FUNCTION_BLOCK "ModularAxis_Speed"   // FB5, LAD
{ S7_Optimized_Access := 'TRUE' }
// stored: MemoryReserve 100, SetENOAutomatically false
   VAR_INPUT
      HomingSensor : Bool;
      Reset : Bool;
      InverterOK : Bool;
      Axis : TO_SpeedAxis;
   END_VAR
   VAR_OUTPUT
      Status : "Status";
   END_VAR
   VAR_IN_OUT
      Execute : Bool;
      PositioningAxis : "S_SpeedAxis";
   END_VAR
   VAR
      State : "s_changeState";
      Delay { S7_SetPoint := 'True'} : "s_TON";
      PowerOff { S7_SetPoint := 'True'} : "s_TON";
      MC_POWER_Instance { ExternalAccessible := 'False'; ExternalVisible := 'False'; ExternalWritable := 'False'} : MC_POWER;
      MC_RESET_Instance { ExternalAccessible := 'False'; ExternalVisible := 'False'; ExternalWritable := 'False'} : MC_RESET;
      MC_HOME_Instance { ExternalAccessible := 'False'; ExternalVisible := 'False'; ExternalWritable := 'False'} : MC_HOME;
      MC_HALT_Instance { ExternalAccessible := 'False'; ExternalVisible := 'False'; ExternalWritable := 'False'} : MC_HALT;
      MC_MOVEJOG_Instance { ExternalAccessible := 'False'; ExternalVisible := 'False'; ExternalWritable := 'False'} : MC_MOVEJOG;
      R_TRIG_Homing { ExternalAccessible := 'False'; ExternalVisible := 'False'; ExternalWritable := 'False'} : R_TRIG;
      R_TRIG_HomeError { ExternalAccessible := 'False'; ExternalVisible := 'False'; ExternalWritable := 'False'} : R_TRIG;
      R_TRIG_HaltError { ExternalAccessible := 'False'; ExternalVisible := 'False'; ExternalWritable := 'False'} : R_TRIG;
      R_TRIG_PowerError { ExternalAccessible := 'False'; ExternalVisible := 'False'; ExternalWritable := 'False'} : R_TRIG;
      R_TRIG_JogError { ExternalAccessible := 'False'; ExternalVisible := 'False'; ExternalWritable := 'False'} : R_TRIG;
      R_TRIG_MoveRelError { ExternalAccessible := 'False'; ExternalVisible := 'False'; ExternalWritable := 'False'} : R_TRIG;
      R_TRIG_ResetError { ExternalAccessible := 'False'; ExternalVisible := 'False'; ExternalWritable := 'False'} : R_TRIG;
      F_TRIG_Inverter { ExternalAccessible := 'False'; ExternalVisible := 'False'; ExternalWritable := 'False'} : F_TRIG;
      Local : Struct
         HomingRequired : Bool;
         prevPosition : LReal;
      END_STRUCT;
   END_VAR
   VAR CONSTANT
      S_IDLE : Int := 10;
      S_HOME : Int := 20;
      S_STOP : Int := 30;
      S_ERROR : Int := 40;
      S_POWER_ON : Int := 50;
      S_MOVE_JOG : Int := 60;
      S_TEST : Int := 100;
      HOMING_ERROR : Word := 16#8000;
      HALT_ERROR : Word := 16#8001;
      POWER_ERROR : Word := 16#8002;
      JOG_ERROR : Word := 16#8003;
      MOVREL_ERROR : Word := 16#8004;
      RESET_ERROR : Word := 16#8005;
   END_VAR
BEGIN

REGION Network 1 (SCL)
   //************************************************************
   //===Author: Mateusz Połojko
   //-----Linkedin: https://pl.linkedin.com/in/mateusz-po%C5%82ojko-52a3541b1
   //-----Github: https://github.com/Bhazel95
   //===Description:
   //-----Motor control as to_speed axis
   //===Customer:
   //-----Apator Powogaz S.A.
   //************************************************************
END_REGION

REGION Network 2
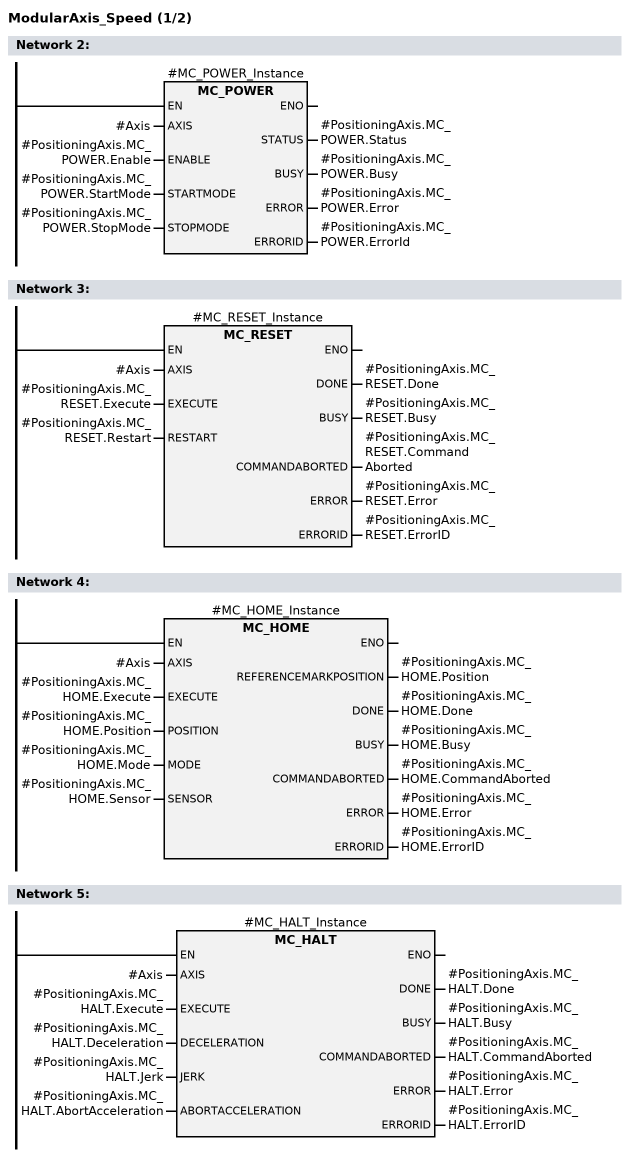
   RUNG wire#powerrail
      #MC_POWER_Instance.MC_POWER(Axis := #Axis, Enable := #PositioningAxis.MC_POWER.Enable, StartMode := #PositioningAxis.MC_POWER.StartMode, StopMode := #PositioningAxis.MC_POWER.StopMode, Status => #PositioningAxis.MC_POWER.Status, Busy => #PositioningAxis.MC_POWER.Busy, Error => #PositioningAxis.MC_POWER.Error, ErrorId => #PositioningAxis.MC_POWER.ErrorId)
   END_RUNG
   // the same network as SCL:
   #MC_POWER_Instance(Axis := #Axis,   // MC_POWER
                      Enable := #PositioningAxis.MC_POWER.Enable,
                      StartMode := #PositioningAxis.MC_POWER.StartMode,
                      StopMode := #PositioningAxis.MC_POWER.StopMode,
                      Status => #PositioningAxis.MC_POWER.Status,
                      Busy => #PositioningAxis.MC_POWER.Busy,
                      Error => #PositioningAxis.MC_POWER.Error,
                      ErrorId => #PositioningAxis.MC_POWER.ErrorId);
END_REGION

REGION Network 3
   RUNG wire#powerrail
      #MC_RESET_Instance.MC_RESET(Axis := #Axis, Execute := #PositioningAxis.MC_RESET.Execute, Restart := #PositioningAxis.MC_RESET.Restart, Done => #PositioningAxis.MC_RESET.Done, Busy => #PositioningAxis.MC_RESET.Busy, CommandAborted => #PositioningAxis.MC_RESET.CommandAborted, Error => #PositioningAxis.MC_RESET.Error, ErrorId => #PositioningAxis.MC_RESET.ErrorID)
   END_RUNG
   // the same network as SCL:
   #MC_RESET_Instance(Axis := #Axis,   // MC_RESET
                      Execute := #PositioningAxis.MC_RESET.Execute,
                      Restart := #PositioningAxis.MC_RESET.Restart,
                      Done => #PositioningAxis.MC_RESET.Done,
                      Busy => #PositioningAxis.MC_RESET.Busy,
                      CommandAborted => #PositioningAxis.MC_RESET.CommandAborted,
                      Error => #PositioningAxis.MC_RESET.Error,
                      ErrorId => #PositioningAxis.MC_RESET.ErrorID);
END_REGION

REGION Network 4
   RUNG wire#powerrail
      #MC_HOME_Instance.MC_HOME(Axis := #Axis, Execute := #PositioningAxis.MC_HOME.Execute, Position := #PositioningAxis.MC_HOME.Position, Mode := #PositioningAxis.MC_HOME.Mode, Sensor := #PositioningAxis.MC_HOME.Sensor, ReferenceMarkPosition => #PositioningAxis.MC_HOME.Position, Done => #PositioningAxis.MC_HOME.Done, Busy => #PositioningAxis.MC_HOME.Busy, CommandAborted => #PositioningAxis.MC_HOME.CommandAborted, Error => #PositioningAxis.MC_HOME.Error, ErrorId => #PositioningAxis.MC_HOME.ErrorID)
   END_RUNG
   // the same network as SCL:
   #MC_HOME_Instance(Axis := #Axis,   // MC_HOME
                     Execute := #PositioningAxis.MC_HOME.Execute,
                     Position := #PositioningAxis.MC_HOME.Position,
                     Mode := #PositioningAxis.MC_HOME.Mode,
                     Sensor := #PositioningAxis.MC_HOME.Sensor,
                     ReferenceMarkPosition => #PositioningAxis.MC_HOME.Position,
                     Done => #PositioningAxis.MC_HOME.Done,
                     Busy => #PositioningAxis.MC_HOME.Busy,
                     CommandAborted => #PositioningAxis.MC_HOME.CommandAborted,
                     Error => #PositioningAxis.MC_HOME.Error,
                     ErrorId => #PositioningAxis.MC_HOME.ErrorID);
END_REGION

REGION Network 5
   RUNG wire#powerrail
      #MC_HALT_Instance.MC_HALT(Axis := #Axis, Execute := #PositioningAxis.MC_HALT.Execute, Deceleration := #PositioningAxis.MC_HALT.Deceleration, Jerk := #PositioningAxis.MC_HALT.Jerk, AbortAcceleration := #PositioningAxis.MC_HALT.AbortAcceleration, Done => #PositioningAxis.MC_HALT.Done, Busy => #PositioningAxis.MC_HALT.Busy, CommandAborted => #PositioningAxis.MC_HALT.CommandAborted, Error => #PositioningAxis.MC_HALT.Error, ErrorId => #PositioningAxis.MC_HALT.ErrorID)
   END_RUNG
   // the same network as SCL:
   #MC_HALT_Instance(Axis := #Axis,   // MC_HALT
                     Execute := #PositioningAxis.MC_HALT.Execute,
                     Deceleration := #PositioningAxis.MC_HALT.Deceleration,
                     Jerk := #PositioningAxis.MC_HALT.Jerk,
                     AbortAcceleration := #PositioningAxis.MC_HALT.AbortAcceleration,
                     Done => #PositioningAxis.MC_HALT.Done,
                     Busy => #PositioningAxis.MC_HALT.Busy,
                     CommandAborted => #PositioningAxis.MC_HALT.CommandAborted,
                     Error => #PositioningAxis.MC_HALT.Error,
                     ErrorId => #PositioningAxis.MC_HALT.ErrorID);
END_REGION

REGION Network 6
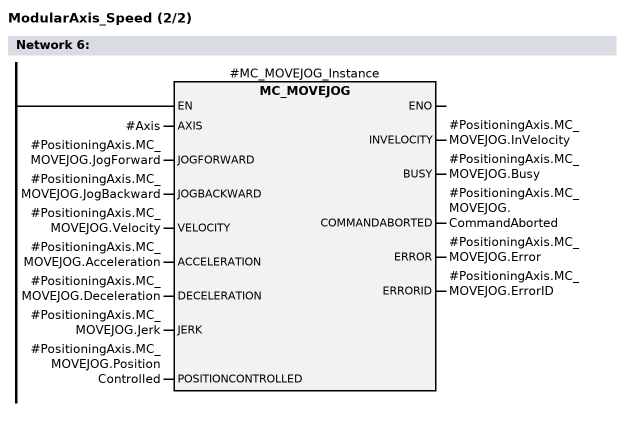
   RUNG wire#powerrail
      #MC_MOVEJOG_Instance.MC_MOVEJOG(Axis := #Axis, JogForward := #PositioningAxis.MC_MOVEJOG.JogForward, JogBackward := #PositioningAxis.MC_MOVEJOG.JogBackward, Velocity := #PositioningAxis.MC_MOVEJOG.Velocity, Acceleration := #PositioningAxis.MC_MOVEJOG.Acceleration, Deceleration := #PositioningAxis.MC_MOVEJOG.Deceleration, Jerk := #PositioningAxis.MC_MOVEJOG.Jerk, PositionControlled := #PositioningAxis.MC_MOVEJOG.PositionControlled, InVelocity => #PositioningAxis.MC_MOVEJOG.InVelocity, Busy => #PositioningAxis.MC_MOVEJOG.Busy, CommandAborted => #PositioningAxis.MC_MOVEJOG.CommandAborted, Error => #PositioningAxis.MC_MOVEJOG.Error, ErrorId => #PositioningAxis.MC_MOVEJOG.ErrorID)
   END_RUNG
   // the same network as SCL:
   #MC_MOVEJOG_Instance(Axis := #Axis,   // MC_MOVEJOG
                        JogForward := #PositioningAxis.MC_MOVEJOG.JogForward,
                        JogBackward := #PositioningAxis.MC_MOVEJOG.JogBackward,
                        Velocity := #PositioningAxis.MC_MOVEJOG.Velocity,
                        Acceleration := #PositioningAxis.MC_MOVEJOG.Acceleration,
                        Deceleration := #PositioningAxis.MC_MOVEJOG.Deceleration,
                        Jerk := #PositioningAxis.MC_MOVEJOG.Jerk,
                        PositionControlled := #PositioningAxis.MC_MOVEJOG.PositionControlled,
                        InVelocity => #PositioningAxis.MC_MOVEJOG.InVelocity,
                        Busy => #PositioningAxis.MC_MOVEJOG.Busy,
                        CommandAborted => #PositioningAxis.MC_MOVEJOG.CommandAborted,
                        Error => #PositioningAxis.MC_MOVEJOG.Error,
                        ErrorId => #PositioningAxis.MC_MOVEJOG.ErrorID);
END_REGION

REGION Network 8 (SCL)
   REGION R/F Trigs
       #F_TRIG_Inverter(CLK := #InverterOK);
       #R_TRIG_HomeError(CLK := #PositioningAxis.MC_HOME.Error);
       #R_TRIG_HaltError(CLK := #PositioningAxis.MC_HALT.Error);
       #R_TRIG_PowerError(CLK := #PositioningAxis.MC_POWER.Error);
       #R_TRIG_JogError(CLK := #PositioningAxis.MC_MOVEJOG.Error);
      // #R_TRIG_MoveRelError(CLK := #PositioningAxis.MC_MOVERELATIVE.Error);
       #R_TRIG_ResetError(CLK := #PositioningAxis.MC_RESET.Error);
       #R_TRIG_Homing(CLK := #HomingSensor);

   END_REGION
   #Delay.PT := T#500MS;
   #Delay.Timer(IN := #Delay.IN,
                PT := #Delay.PT);
   #PowerOff.PT := T#180S;
   #PowerOff.Timer(IN := #PowerOff.IN,
                   PT := #PowerOff.PT);

   CASE #State.state OF
       #S_IDLE:
           //Funkcja wejścia
           IF #State.inputFlag AND NOT #State.outputFlag THEN
               #Execute := FALSE;
               #State.name := 'IDLE';
               #Status.Busy := FALSE;
               #Status.Ready := TRUE;
               // #Status.Done := FALSE;
               #Status.Error := FALSE;
               #PowerOff.IN := TRUE;
           END_IF;

           //Funkcja cykliczna
           IF NOT #State.inputFlag AND NOT #State.outputFlag THEN
               IF #PowerOff.Timer.Q THEN
                   #PositioningAxis.MC_POWER.Enable := FALSE;
               END_IF;
               IF #Reset THEN
                   // Statement section IF
                   ;
               END_IF;


               IF #Execute THEN
                   IF #PositioningAxis.MC_POWER.Status THEN
                       "changeState"(newState := #S_MOVE_JOG,
                                     Data := #State);
                   ELSE
                       #PositioningAxis.MC_POWER.Enable := FALSE;
                       "changeState"(newState := #S_POWER_ON,
                                     Data := #State);
                   END_IF;
               END_IF;
               IF #PositioningAxis.MC_MOVEJOG.JogForward OR #PositioningAxis.MC_MOVEJOG.JogBackward THEN
                   #Status.Done := FALSE;
                   #Status.Busy := TRUE;
                   //#Local.HomingRequired := TRUE;
               END_IF;
           END_IF;

           //Funkcja wyjściowa 
           IF #State.outputFlag THEN
               #PowerOff.IN := FALSE;
               #Status.Busy := TRUE;
           END_IF;

       #S_HOME:
           //Funkcja wejścia
           IF #State.inputFlag AND NOT #State.outputFlag THEN
               #State.name := 'HOMING';
               #Status.Busy := TRUE;
               #Status.Ready := FALSE;
               #Status.Done := FALSE;
               #Status.Error := FALSE;
               #PositioningAxis.MC_HOME.Mode := 8;
               #PositioningAxis.MC_HOME.Execute := TRUE;
           END_IF;

           //Funkcja cykliczna
           IF NOT #State.inputFlag AND NOT #State.outputFlag THEN
               IF #PositioningAxis.MC_HOME.Done THEN
                   #Local.HomingRequired := FALSE;
                   #Status.Done := TRUE;
                   "changeState"(newState := #S_IDLE,
                                 Data := #State);
               END_IF;
           END_IF;

           //Funkcja wyjściowa 
           IF #State.outputFlag THEN
               #PositioningAxis.MC_HOME.Execute := FALSE;
           END_IF;

       #S_ERROR:
           //Funkcja wejścia
           IF #State.inputFlag AND NOT #State.outputFlag THEN
               #State.name := 'ERROR';
               #Status.Busy := FALSE;
               #Status.Ready := FALSE;
               #Status.Done := FALSE;
               #Status.Error := TRUE;
               //#Local.HomingRequired := TRUE;
               #PositioningAxis.MC_HOME.Execute := FALSE;
               #PositioningAxis.MC_POWER.Enable := FALSE;
              // #PositioningAxis.MC_MOVERELATIVE.Execute := FALSE;
               #PositioningAxis.MC_HALT.Execute := FALSE;
               #PositioningAxis.MC_RESET.Execute := FALSE;
               #PositioningAxis.MC_MOVEJOG.JogBackward := FALSE;
               #PositioningAxis.MC_MOVEJOG.JogForward := FALSE;
           END_IF;

           //Funkcja cykliczna
           IF NOT #State.inputFlag AND NOT #State.outputFlag THEN
               IF #Reset THEN
                   // #MC_RESET_Instance.Restart := FALSE;
                   #PositioningAxis.MC_RESET.Execute := TRUE;
               END_IF;
               IF #PositioningAxis.MC_RESET.Done AND #InverterOK THEN
                   "changeState"(newState := #S_POWER_ON,
                                 Data := #State);
               END_IF;
           END_IF;

           //Funkcja wyjściowa 
           IF #State.outputFlag THEN
               #Status.Error := FALSE;
               #Status.Busy := TRUE;
               #PositioningAxis.MC_RESET.Execute := FALSE;
           END_IF;

       #S_POWER_ON:
           //Funkcja wejścia
           IF #State.inputFlag AND NOT #State.outputFlag THEN
               #State.name := 'ERROR';
               #Status.Busy := TRUE;
               #Status.Ready := FALSE;
               #Status.Done := FALSE;
               #Status.Error := FALSE;
               #PositioningAxis.MC_POWER.Enable := TRUE;
           END_IF;

           //Funkcja cykliczna
           IF NOT #State.inputFlag AND NOT #State.outputFlag THEN
               IF #PositioningAxis.MC_POWER.Status THEN
                   "changeState"(newState := #S_IDLE,
                                 Data := #State);
               END_IF;
           END_IF;

           //Funkcja wyjściowa 
           IF #State.outputFlag THEN
               ;
           END_IF;

       #S_MOVE_JOG:
           //Funkcja wejścia
           IF #State.inputFlag AND NOT #State.outputFlag THEN
               #State.name := 'MOVING';
               #Status.Busy := TRUE;
               #Status.Ready := FALSE;
               #Status.Done := FALSE;
               #Status.Error := FALSE;
               //#Local.prevPosition := #Axis.ActualPosition;
               #PositioningAxis.MC_MOVEJOG.Acceleration := 0.3;
               #PositioningAxis.MC_MOVEJOG.Deceleration := 0.7;
               #PositioningAxis.MC_MOVEJOG.Velocity := 0.15;
               #PositioningAxis.MC_MOVEJOG.JogBackward := FALSE;
               #PositioningAxis.MC_MOVEJOG.JogForward := TRUE;
               #Delay.IN := FALSE;
           END_IF;

           //Funkcja cykliczna
           IF NOT #State.inputFlag AND NOT #State.outputFlag THEN
               IF #R_TRIG_Homing.Q THEN
                   #Status.Done := TRUE;
                   #PositioningAxis.MC_MOVEJOG.JogBackward := FALSE;
                   #PositioningAxis.MC_MOVEJOG.JogForward := FALSE;
                   #Delay.IN := TRUE;
               END_IF;
               IF #Delay.Timer.Q THEN

                   "changeState"(newState := #S_IDLE,
                                 Data := #State);
               END_IF;

           END_IF;

           //Funkcja wyjściowa 
           IF #State.outputFlag THEN
               #Delay.IN := FALSE;
           END_IF;

       #S_TEST:
           ;
   END_CASE;

   IF #R_TRIG_HomeError.Q THEN
       #Status.ErrorStatus := #HOMING_ERROR;
       "changeState"(newState := #S_ERROR,
                     Data := #State);
   ELSIF #R_TRIG_HaltError.Q THEN
       #Status.ErrorStatus := #HALT_ERROR;
       "changeState"(newState := #S_ERROR,
                     Data := #State);
   ELSIF #R_TRIG_JogError.Q THEN
       #Status.ErrorStatus := #JOG_ERROR;
       "changeState"(newState := #S_ERROR,
                     Data := #State);
   ELSIF #R_TRIG_MoveRelError.Q THEN
       #Status.ErrorStatus := #MOVREL_ERROR;
       "changeState"(newState := #S_ERROR,
                     Data := #State);
   ELSIF #R_TRIG_PowerError.Q THEN
       #Status.ErrorStatus := #POWER_ERROR;
       "changeState"(newState := #S_ERROR,
                     Data := #State);
   ELSIF #R_TRIG_ResetError.Q THEN
       #Status.ErrorStatus := #RESET_ERROR;
       "changeState"(newState := #S_ERROR,
                     Data := #State);
   END_IF;

   IF #F_TRIG_Inverter.Q THEN
       "changeState"(newState := #S_ERROR,
                     Data := #State);
   END_IF;

   IF NOT "DEV_7".Convoyer.Modular_A.Sensors.JogBack THEN
       #PositioningAxis.MC_MOVEJOG.JogBackward := FALSE;
   END_IF;

   REGION Change state
       IF #State.inputFlag AND NOT #State.outputFlag THEN
           #State.inputFlag := FALSE;
       END_IF;
       #State.outputFlag := FALSE;
   END_REGION
END_REGION
END_FUNCTION_BLOCK

FUNCTION "FC_008_OPC" : Void
{ S7_Optimized_Access := 'TRUE' }
VERSION : 0.1

BEGIN
END_FUNCTION

FUNCTION "FC_09_HMI" : Void
{ S7_Optimized_Access := 'TRUE' }
VERSION : 0.1

BEGIN
	//************************************************************
	//===Author: Mateusz Połojko
	//-----Linkedin: https://pl.linkedin.com/in/mateusz-po%C5%82ojko-52a3541b1
	//-----Github: https://github.com/Bhazel95
	//===Description:
	//-----HMI assigments
	//===Customer:
	//-----Apator Powogaz S.A.
	//************************************************************
	
	REGION Camera state  
	    "DEV_7".Convoyer.Modular_A.HMI.Camera.State := "ModularConvoyer_7A_DB".CameraConnectionTCP_Instance.State.name;
	    "DEV_7".Convoyer.Modular_B.HMI.Camera.State := "ModularConvoyer_7B_DB".CameraConnectionTCP_Instance.State.name;
	    "DEV_10".Convoyer.Modular_A.HMI.Camera.State := "ModularConvoyer_10A_DB".CameraConnectionTCP_Instance.State.name;
	END_REGION
	
END_FUNCTION

FUNCTION "FC_010_Outputs" : Void
{ S7_Optimized_Access := 'TRUE' }
VERSION : 0.1

BEGIN
	//************************************************************
	//===Author: Mateusz Połojko
	//-----Linkedin: https://pl.linkedin.com/in/mateusz-po%C5%82ojko-52a3541b1
	//-----Github: https://github.com/Bhazel95
	//===Description:
	//-----Hardware output assigment
	//===Customer:
	//-----Apator Powogaz S.A.
	//************************************************************
	
	REGION 7A
	    REGION Button box left
	        "7A_BUTTON_LIGHT_START_1" := "DEV_7".Convoyer.Modular_A.ButtonControl.ButtonBoxLeft.LightStart;
	        "7A_BUTTON_LIGHT_RESET_1" := "DEV_7".Convoyer.Modular_A.ButtonControl.ButtonBoxLeft.LightReset;
	        "7A_BUTTON_LIGHT_STOP_1" := "DEV_7".Convoyer.Modular_A.ButtonControl.ButtonBoxLeft.LightStop;
	        "7A_BUTTON_LIGHT_ESTOP_1" := NOT "7A_ESTOP_1";
	    END_REGION
	    REGION Button box right
	        "7A_BUTTON_LIGHT_START_2" := "DEV_7".Convoyer.Modular_A.ButtonControl.ButtonBoxRight.LightStart;
	        "7A_BUTTON_LIGHT_RESET_2" := "DEV_7".Convoyer.Modular_A.ButtonControl.ButtonBoxRight.LightReset;
	        "7A_BUTTON_LIGHT_STOP_2" := "DEV_7".Convoyer.Modular_A.ButtonControl.ButtonBoxRight.LightStop;
	        "7A_BUTTON_LIGHT_ESTOP_2" := NOT "7A_ESTOP_2";
	    END_REGION
	    REGION Lights    
	        "7A_LIGHTS_BUZZER_1" := "DEV_7".Convoyer.Modular_A.Lights.Blue;
	        "7A_LIGHTS_GREEN_1" := "DEV_7".Convoyer.Modular_A.Lights.Green;
	        "7A_LIGHTS_RED_1" := "DEV_7".Convoyer.Modular_A.Lights.Red;
	        "7A_LIGHTS_ORANGE_1" := "DEV_7".Convoyer.Modular_A.Lights.Orange;
	    END_REGION
	    REGION Pneumatics
	        "7A_VALVE_IN_1" := "DEV_7".Convoyer.Modular_A.Pneumatics.Stamping.Coils.In;
	        "7A_VALVE_OUT_1" := "DEV_7".Convoyer.Modular_A.Pneumatics.Stamping.Coils.Out;
	        
	        "7A_VALVE_IN_2" := "DEV_7".Convoyer.Modular_A.Pneumatics.Valve.Coils.In;
	        "7A_VALVE_OUT_2" := "DEV_7".Convoyer.Modular_A.Pneumatics.Valve.Coils.Out;
	        
	        IF "DEV_7".Convoyer.Modular_A.Safety.SafetyOK AND "DEV_7".Convoyer.Modular_A.Sensors.Span THEN
	            "DEV_7".Convoyer.Modular_A.Pneumatics.IVT.Sensor.Scaled.SetNorm := NORM_X(MIN := 0, VALUE := "DEV_7".Convoyer.Modular_A.Pneumatics.IVT.Sensor.Analog.SetValue, MAX := 7);
	            "7A_IVT_OutputSignal_1" := SCALE_X(MIN := 0, VALUE := "DEV_7".Convoyer.Modular_A.Pneumatics.IVT.Sensor.Scaled.SetNorm, MAX := 32767);
	        ELSE
	            "DEV_7".Convoyer.Modular_A.Pneumatics.IVT.Sensor.Scaled.SetNorm := NORM_X(MIN := 0.0, VALUE := 0.0, MAX := 7);
	            "7A_IVT_OutputSignal_1" := SCALE_X(MIN := 0, VALUE := "DEV_7".Convoyer.Modular_A.Pneumatics.IVT.Sensor.Scaled.SetNorm, MAX := 32767);
	        END_IF;
	    END_REGION
	END_REGION
	REGION 7B
	    REGION Button box left
	        "7B_BUTTON_LIGHT_START_1" := "DEV_7".Convoyer.Modular_B.ButtonControl.ButtonBoxLeft.LightStart;
	        "7B_BUTTON_LIGHT_RESET_1" := "DEV_7".Convoyer.Modular_B.ButtonControl.ButtonBoxLeft.LightReset;
	        "7B_BUTTON_LIGHT_STOP_1" := "DEV_7".Convoyer.Modular_B.ButtonControl.ButtonBoxLeft.LightStop;
	        "7B_BUTTON_LIGHT_ESTOP_1" := NOT "7B_ESTOP_1";
	    END_REGION
	    REGION Button box right
	        "7B_BUTTON_LIGHT_START_2" := "DEV_7".Convoyer.Modular_B.ButtonControl.ButtonBoxRight.LightStart;
	        "7B_BUTTON_LIGHT_RESET_2" := "DEV_7".Convoyer.Modular_B.ButtonControl.ButtonBoxRight.LightReset;
	        "7B_BUTTON_LIGHT_STOP_2" := "DEV_7".Convoyer.Modular_B.ButtonControl.ButtonBoxRight.LightStop;
	        "7B_BUTTON_LIGHT_ESTOP_2" := NOT "7B_ESTOP_2";
	    END_REGION
	    REGION Lights    
	        "7B_LIGHTS_BUZZER_1" := "DEV_7".Convoyer.Modular_B.Lights.Blue;
	        "7B_LIGHTS_GREEN_1" := "DEV_7".Convoyer.Modular_B.Lights.Green;
	        "7B_LIGHTS_RED_1" := "DEV_7".Convoyer.Modular_B.Lights.Red;
	        "7B_LIGHTS_ORANGE_1" := "DEV_7".Convoyer.Modular_B.Lights.Orange;
	    END_REGION
	    REGION Pneumatics
	        "7B_VALVE_IN_2" := "DEV_7".Convoyer.Modular_B.Pneumatics.Stamping.Coils.In;
	        "7B_VALVE_OUT_2" := "DEV_7".Convoyer.Modular_B.Pneumatics.Stamping.Coils.Out;
	        
	        "7B_VALVE_IN_1" := "DEV_7".Convoyer.Modular_B.Pneumatics.Valve.Coils.In;
	        "7B_VALVE_OUT_1" := "DEV_7".Convoyer.Modular_B.Pneumatics.Valve.Coils.Out;
	        
	        IF "DEV_7".Convoyer.Modular_B.Safety.SafetyOK AND "DEV_7".Convoyer.Modular_B.Sensors.Span THEN
	            "DEV_7".Convoyer.Modular_B.Pneumatics.IVT.Sensor.Scaled.SetNorm := NORM_X(MIN := 0, VALUE := "DEV_7".Convoyer.Modular_B.Pneumatics.IVT.Sensor.Analog.SetValue, MAX := 7);
	            "7B_IVT_OutputSignal_1" := SCALE_X(MIN := 0, VALUE := "DEV_7".Convoyer.Modular_B.Pneumatics.IVT.Sensor.Scaled.SetNorm, MAX := 32767);
	        ELSE
	            "DEV_7".Convoyer.Modular_B.Pneumatics.IVT.Sensor.Scaled.SetNorm := NORM_X(MIN := 0.0, VALUE := 0.0, MAX := 7);
	            "7B_IVT_OutputSignal_1" := SCALE_X(MIN := 0, VALUE := "DEV_7".Convoyer.Modular_B.Pneumatics.IVT.Sensor.Scaled.SetNorm, MAX := 32767);
	        END_IF;
	    END_REGION
	END_REGION
	REGION Main Cabinet
	    "7_BUTTON_LIGHT_RESET_6" := "DEV_7".Convoyer.Modular_A.ButtonControl.CabinetBox.LightReset OR "DEV_7".Convoyer.Modular_B.ButtonControl.CabinetBox.LightReset;
	    "7_BUTTON_LIGHT_ESTOP_6" := NOT "7_ESTOP";
	END_REGION
	REGION 24V Main Cabinet
	    "7AB_24V_OK" := "7_24V_OK";
	END_REGION
	
	
	REGION 10A
	    REGION Button box left
	        "10A_BUTTON_LIGHT_START_1" := "DEV_10".Convoyer.Modular_A.ButtonControl.ButtonBoxLeft.LightStart;
	        "10A_BUTTON_LIGHT_RESET_1" := "DEV_10".Convoyer.Modular_A.ButtonControl.ButtonBoxLeft.LightReset;
	        "10A_BUTTON_LIGHT_STOP_1" := "DEV_10".Convoyer.Modular_A.ButtonControl.ButtonBoxLeft.LightStop;
	        "10A_BUTTON_LIGHT_ESTOP_1" := NOT "10A_ESTOP_1";
	    END_REGION
	    REGION Button box right
	        "10A_BUTTON_LIGHT_START_2" := "DEV_10".Convoyer.Modular_A.ButtonControl.ButtonBoxRight.LightStart;
	        "10A_BUTTON_LIGHT_RESET_2" := "DEV_10".Convoyer.Modular_A.ButtonControl.ButtonBoxRight.LightReset;
	        "10A_BUTTON_LIGHT_STOP_2" := "DEV_10".Convoyer.Modular_A.ButtonControl.ButtonBoxRight.LightStop;
	        "10A_BUTTON_LIGHT_ESTOP_2" := NOT "10A_ESTOP_2";
	    END_REGION
	    REGION Lights    
	        "10A_LIGHTS_BUZZER_1" := "DEV_10".Convoyer.Modular_A.Lights.Blue;
	        "10A_LIGHTS_GREEN_1" := "DEV_10".Convoyer.Modular_A.Lights.Green;
	        "10A_LIGHTS_RED_1" := "DEV_10".Convoyer.Modular_A.Lights.Red;
	        "10A_LIGHTS_ORANGE_1" := "DEV_10".Convoyer.Modular_A.Lights.Orange;
	    END_REGION
	    REGION Pneumatics
	        "10A_VALVE_IN_1" := "DEV_10".Convoyer.Modular_A.Pneumatics.Stamping.Coils.In;
	        "10A_VALVE_OUT_1" := "DEV_10".Convoyer.Modular_A.Pneumatics.Stamping.Coils.Out;
	        
	        "10A_VALVE_IN_2" := "DEV_10".Convoyer.Modular_A.Pneumatics.Valve.Coils.In;
	        "10A_VALVE_OUT_2" := "DEV_10".Convoyer.Modular_A.Pneumatics.Valve.Coils.Out;
	        
	        IF "DEV_10".Convoyer.Modular_A.Safety.SafetyOK AND "DEV_10".Convoyer.Modular_A.Sensors.Span THEN
	            "DEV_10".Convoyer.Modular_A.Pneumatics.IVT.Sensor.Scaled.SetNorm := NORM_X(MIN := 0, VALUE := "DEV_10".Convoyer.Modular_A.Pneumatics.IVT.Sensor.Analog.SetValue, MAX := 7);
	            "10A_IVT_OutputSignal_1" := SCALE_X(MIN := 0, VALUE := "DEV_10".Convoyer.Modular_A.Pneumatics.IVT.Sensor.Scaled.SetNorm, MAX := 32767);
	        ELSE
	            "DEV_10".Convoyer.Modular_A.Pneumatics.IVT.Sensor.Scaled.SetNorm := NORM_X(MIN := 0.0, VALUE := 0.0, MAX := 7);
	            "10A_IVT_OutputSignal_1" := SCALE_X(MIN := 0, VALUE := "DEV_10".Convoyer.Modular_A.Pneumatics.IVT.Sensor.Scaled.SetNorm, MAX := 32767);
	        END_IF;
	    END_REGION
	END_REGION
	REGION 10 Cabinet
	    //dla 10b dodac or 10b
	    "10_BUTTON_LIGHT_RESET_6" := "DEV_10".Convoyer.Modular_A.ButtonControl.CabinetBox.LightReset;
	    "10_BUTTON_LIGHT_ESTOP_6" := NOT "10_ESTOP";
	END_REGION
	//Do zmiany
	REGION 24V 10 Cabinet  
	    "10AB_24V_OK" := TRUE;
	END_REGION
	
END_FUNCTION

FUNCTION_BLOCK "CabinetDiagReset_10"   // FB13, F_LAD
{ S7_Optimized_Access := 'TRUE' }
   VAR_INPUT
      RESET : Bool;
   END_VAR
BEGIN

REGION Network 1: 1=Acknowledgment for reintegration
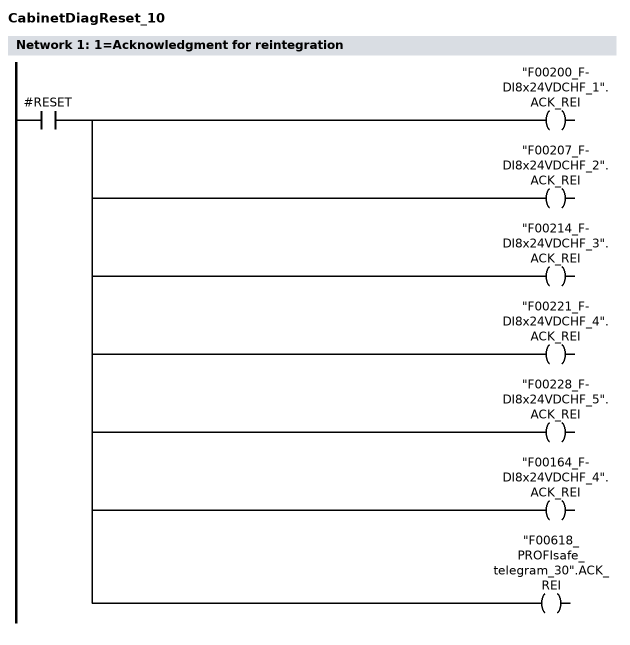
   RUNG wire#powerrail
      Contact( #RESET )
      wire#w1
      Coil( "F00200_F-DI8x24VDCHF_1".ACK_REI )
   END_RUNG
   RUNG wire#w1
      Coil( "F00207_F-DI8x24VDCHF_2".ACK_REI )
   END_RUNG
   RUNG wire#w1
      Coil( "F00214_F-DI8x24VDCHF_3".ACK_REI )
   END_RUNG
   RUNG wire#w1
      Coil( "F00221_F-DI8x24VDCHF_4".ACK_REI )
   END_RUNG
   RUNG wire#w1
      Coil( "F00228_F-DI8x24VDCHF_5".ACK_REI )
   END_RUNG
   RUNG wire#w1
      Coil( "F00164_F-DI8x24VDCHF_4".ACK_REI )
   END_RUNG
   RUNG wire#w1
      Coil( "F00618_PROFIsafe_telegram_30".ACK_REI )
   END_RUNG
   // the same network as SCL:
   "F00200_F-DI8x24VDCHF_1".ACK_REI := #RESET;
   "F00207_F-DI8x24VDCHF_2".ACK_REI := #RESET;
   "F00214_F-DI8x24VDCHF_3".ACK_REI := #RESET;
   "F00221_F-DI8x24VDCHF_4".ACK_REI := #RESET;
   "F00228_F-DI8x24VDCHF_5".ACK_REI := #RESET;
   "F00164_F-DI8x24VDCHF_4".ACK_REI := #RESET;
   "F00618_PROFIsafe_telegram_30".ACK_REI := #RESET;
END_REGION
END_FUNCTION_BLOCK

FUNCTION_BLOCK "Convoyer7"   // FB6, F_LAD
{ S7_Optimized_Access := 'TRUE' }
   VAR_INPUT
      InverterStatus : "LDrvSafe_typeSinaTlg30Status";
      ESTOP : Bool;
      LIGHT_CURTAIN : Bool;
      PROCES_STAMPING : Bool;
      DOOR : Bool;
      FRQ_FEEDBACK : Bool;
      RESET : Bool;
   END_VAR
   VAR_OUTPUT
      InverterControl : "LDrvSafe_typeSinaTlg30Control";
      SAFETY_OK : Bool;
      INVERTER_OK : Bool;
      FRQ_NOK : Bool;
      REQ_RESET_ESTOP : Bool;
      SAFETY_VALVE : Bool;
   END_VAR
   VAR
      ESTOP_ON : Bool;
      INVERTER_FAULT : Bool;
      ESTOP1_Instance : ESTOP1;
      LDrvSafe_SinaTlg30Control_Instance : "LDrvSafe_SinaTlg30Control";
      LDrvSafe_SinaTlg30Status_Instance : "LDrvSafe_SinaTlg30Status";
   END_VAR
BEGIN

REGION Network 1
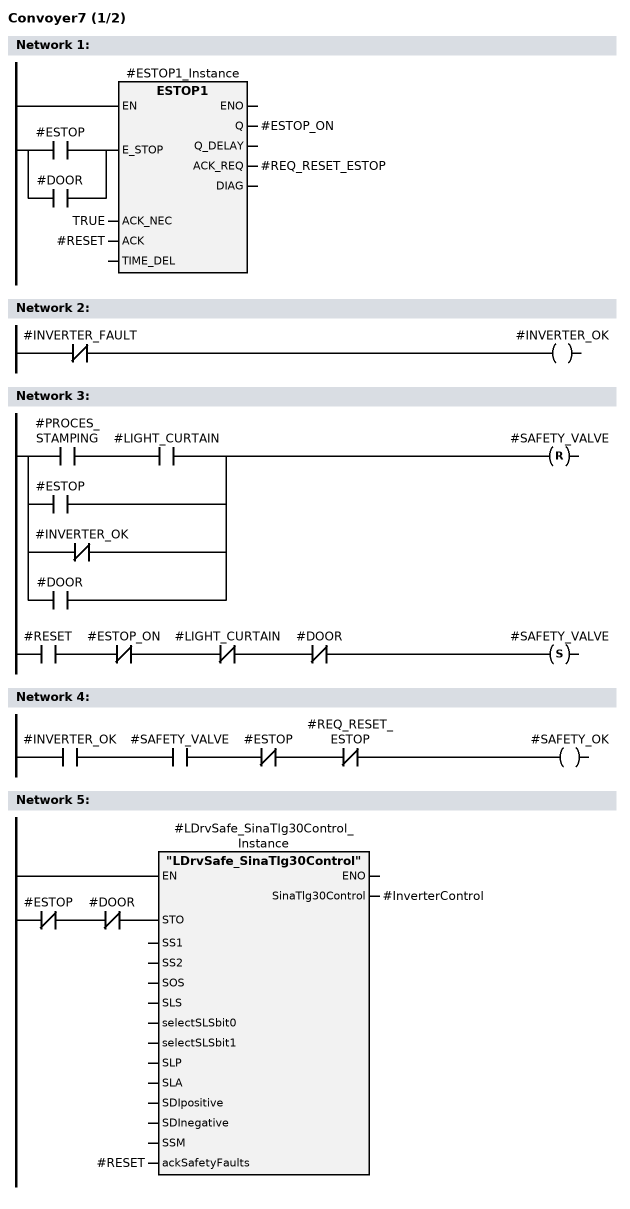
   RUNG wire#powerrail
      #ESTOP1_Instance.ESTOP1(E_STOP := wire#w1, ACK_NEC := TRUE, ACK := #RESET, TIME_DEL :=, Q => #ESTOP_ON, Q_DELAY =>, ACK_REQ => #REQ_RESET_ESTOP, DIAG =>)
   END_RUNG
   RUNG wire#powerrail
      Contact( #ESTOP )
   END_RUNG wire#w1
   RUNG wire#powerrail
      Contact( #DOOR )
   END_RUNG wire#w1
   // the same network as SCL:
   #ESTOP1_Instance(E_STOP := #ESTOP OR #DOOR,   // ESTOP1
                    ACK_NEC := TRUE,
                    ACK := #RESET,
                    Q => #ESTOP_ON,
                    ACK_REQ => #REQ_RESET_ESTOP);
END_REGION

REGION Network 2
   RUNG wire#powerrail
      I_Contact( #INVERTER_FAULT )
      Coil( #INVERTER_OK )
   END_RUNG
   // the same network as SCL:
   #INVERTER_OK := NOT #INVERTER_FAULT;
END_REGION

REGION Network 3
   RUNG wire#powerrail
      Contact( #PROCES_STAMPING )
      Contact( #LIGHT_CURTAIN )
      wire#w1
      R_Coil( #SAFETY_VALVE )
   END_RUNG
   RUNG wire#powerrail
      Contact( #ESTOP )
   END_RUNG wire#w1
   RUNG wire#powerrail
      I_Contact( #INVERTER_OK )
   END_RUNG wire#w1
   RUNG wire#powerrail
      Contact( #DOOR )
   END_RUNG wire#w1
   RUNG wire#powerrail
      Contact( #RESET )
      I_Contact( #ESTOP_ON )
      I_Contact( #LIGHT_CURTAIN )
      I_Contact( #DOOR )
      S_Coil( #SAFETY_VALVE )
   END_RUNG
   // the same network as SCL:
   IF (#PROCES_STAMPING AND #LIGHT_CURTAIN) OR #ESTOP OR NOT #INVERTER_OK OR #DOOR THEN
       #SAFETY_VALVE := FALSE;
   END_IF;
   IF #RESET AND NOT #ESTOP_ON AND NOT #LIGHT_CURTAIN AND NOT #DOOR THEN #SAFETY_VALVE := TRUE; END_IF;
END_REGION

REGION Network 4
   RUNG wire#powerrail
      Contact( #INVERTER_OK )
      Contact( #SAFETY_VALVE )
      I_Contact( #ESTOP )
      I_Contact( #REQ_RESET_ESTOP )
      Coil( #SAFETY_OK )
   END_RUNG
   // the same network as SCL:
   #SAFETY_OK := #INVERTER_OK AND #SAFETY_VALVE AND NOT #ESTOP AND NOT #REQ_RESET_ESTOP;
END_REGION

REGION Network 5
   RUNG wire#powerrail
      #LDrvSafe_SinaTlg30Control_Instance(STO := wire#w1, SS1 :=, SS2 :=, SOS :=, SLS :=, selectSLSbit0 :=, selectSLSbit1 :=, SLP :=, SLA :=, SDIpositive :=, SDInegative :=, SSM :=, ackSafetyFaults := #RESET, SinaTlg30Control => #InverterControl)
   END_RUNG
   RUNG wire#powerrail
      I_Contact( #ESTOP )
      I_Contact( #DOOR )
   END_RUNG wire#w1
   // the same network as SCL:
   #LDrvSafe_SinaTlg30Control_Instance(STO := NOT #ESTOP AND NOT #DOOR,   // "LDrvSafe_SinaTlg30Control"
                           ackSafetyFaults := #RESET,
                           SinaTlg30Control => #InverterControl);
END_REGION

REGION Network 6
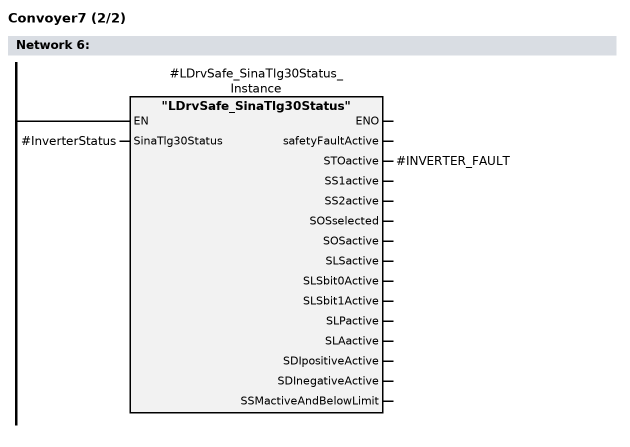
   RUNG wire#powerrail
      #LDrvSafe_SinaTlg30Status_Instance(SinaTlg30Status := #InverterStatus, safetyFaultActive =>, STOactive => #INVERTER_FAULT, SS1active =>, SS2active =>, SOSselected =>, SOSactive =>, SLSactive =>, SLSbit0Active =>, SLSbit1Active =>, SLPactive =>, SLAactive =>, SDIpositiveActive =>, SDInegativeActive =>, SSMactiveAndBelowLimit =>)
   END_RUNG
   // the same network as SCL:
   #LDrvSafe_SinaTlg30Status_Instance(SinaTlg30Status := #InverterStatus, STOactive => #INVERTER_FAULT);   // "LDrvSafe_SinaTlg30Status"
END_REGION
END_FUNCTION_BLOCK

FUNCTION_BLOCK "MainCabinetDiagReset"   // FB12, F_LAD
{ S7_Optimized_Access := 'TRUE' }
   VAR_INPUT
      RESET : Bool;
   END_VAR
BEGIN

REGION Network 1: 1=Acknowledgment for reintegration
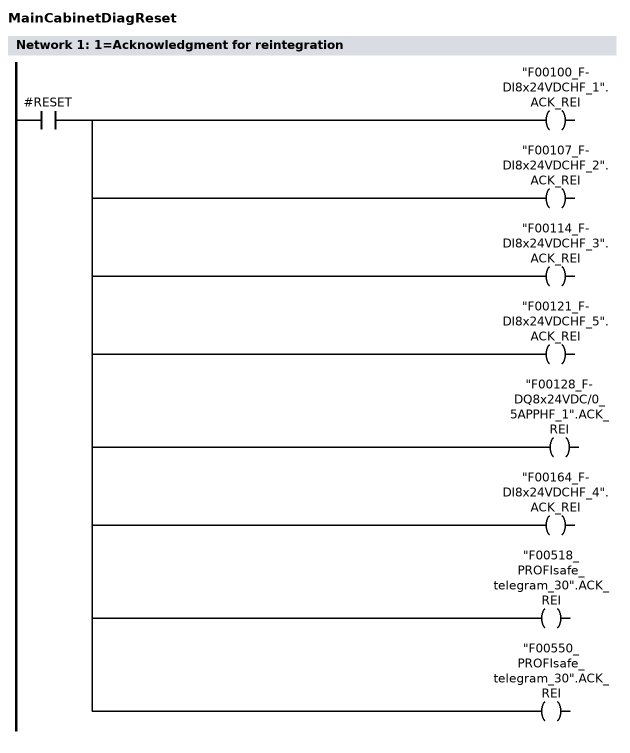
   RUNG wire#powerrail
      Contact( #RESET )
      wire#w1
      Coil( "F00100_F-DI8x24VDCHF_1".ACK_REI )
   END_RUNG
   RUNG wire#w1
      Coil( "F00107_F-DI8x24VDCHF_2".ACK_REI )
   END_RUNG
   RUNG wire#w1
      Coil( "F00114_F-DI8x24VDCHF_3".ACK_REI )
   END_RUNG
   RUNG wire#w1
      Coil( "F00121_F-DI8x24VDCHF_5".ACK_REI )
   END_RUNG
   RUNG wire#w1
      Coil( "F00128_F-DQ8x24VDC/0_5APPHF_1".ACK_REI )
   END_RUNG
   RUNG wire#w1
      Coil( "F00164_F-DI8x24VDCHF_4".ACK_REI )
   END_RUNG
   RUNG wire#w1
      Coil( "F00518_PROFIsafe_telegram_30".ACK_REI )
   END_RUNG
   RUNG wire#w1
      Coil( "F00550_PROFIsafe_telegram_30".ACK_REI )
   END_RUNG
   // the same network as SCL:
   "F00100_F-DI8x24VDCHF_1".ACK_REI := #RESET;
   "F00107_F-DI8x24VDCHF_2".ACK_REI := #RESET;
   "F00114_F-DI8x24VDCHF_3".ACK_REI := #RESET;
   "F00121_F-DI8x24VDCHF_5".ACK_REI := #RESET;
   "F00128_F-DQ8x24VDC/0_5APPHF_1".ACK_REI := #RESET;
   "F00164_F-DI8x24VDCHF_4".ACK_REI := #RESET;
   "F00518_PROFIsafe_telegram_30".ACK_REI := #RESET;
   "F00550_PROFIsafe_telegram_30".ACK_REI := #RESET;
END_REGION
END_FUNCTION_BLOCK

FUNCTION_BLOCK "Main_Safety_RTG1"   // FB1, F_LAD
{ S7_Optimized_Access := 'TRUE' }
// stored: AutoNumber false
   VAR
      Convoyer7A_Instance : "Convoyer7";
      MainCabinetDiagReset_Instance : "MainCabinetDiagReset";
      Convoyer7B_Instance : "Convoyer7";
      CabinetDiagReset_10_Instance : "CabinetDiagReset_10";
      Convoyer10A_DB : "Convoyer7";
   END_VAR
BEGIN

REGION Network 1
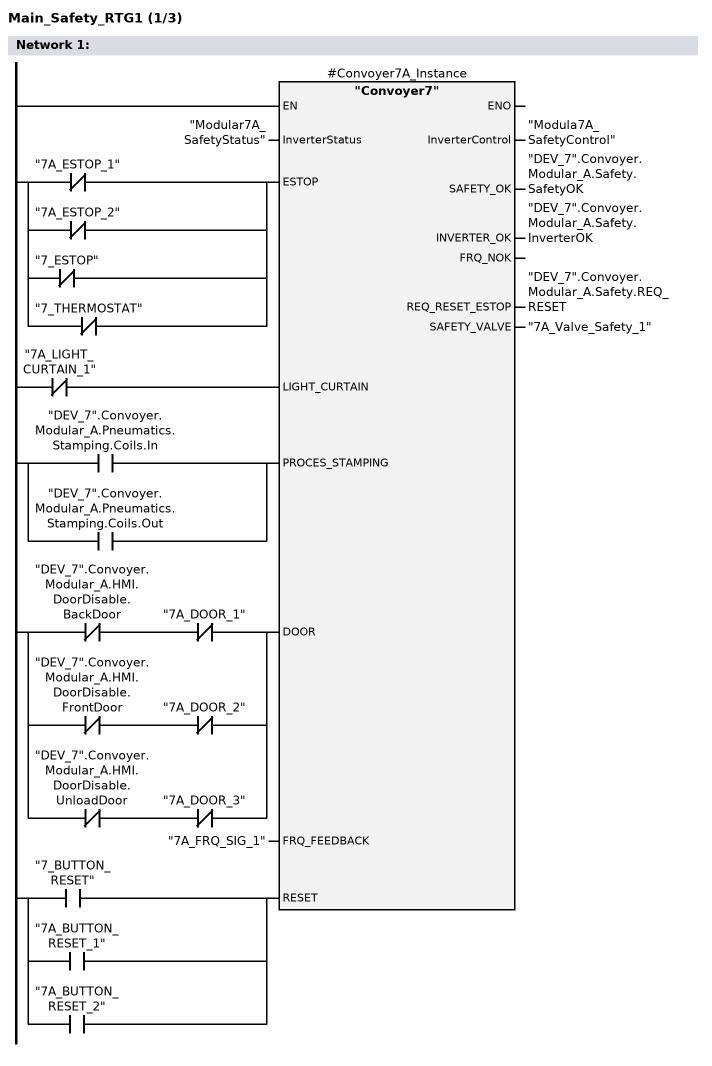
   RUNG wire#powerrail
      #Convoyer7A_Instance(ESTOP := wire#w1, LIGHT_CURTAIN := wire#w2, PROCES_STAMPING := wire#w3, DOOR := wire#w4, RESET := wire#w5, InverterStatus := "Modular7A_SafetyStatus", FRQ_FEEDBACK := "7A_FRQ_SIG_1", InverterControl => "Modula7A_SafetyControl", SAFETY_OK => "DEV_7".Convoyer.Modular_A.Safety.SafetyOK, INVERTER_OK => "DEV_7".Convoyer.Modular_A.Safety.InverterOK, FRQ_NOK =>, REQ_RESET_ESTOP => "DEV_7".Convoyer.Modular_A.Safety.REQ_RESET, SAFETY_VALVE => "7A_Valve_Safety_1")
   END_RUNG
   RUNG wire#powerrail
      I_Contact( "7A_ESTOP_1" )
   END_RUNG wire#w1
   RUNG wire#powerrail
      I_Contact( "7A_ESTOP_2" )
   END_RUNG wire#w1
   RUNG wire#powerrail
      I_Contact( "7_ESTOP" )
   END_RUNG wire#w1
   RUNG wire#powerrail
      I_Contact( "7_THERMOSTAT" )
   END_RUNG wire#w1
   RUNG wire#powerrail
      I_Contact( "7A_LIGHT_CURTAIN_1" )
   END_RUNG wire#w2
   RUNG wire#powerrail
      Contact( "DEV_7".Convoyer.Modular_A.Pneumatics.Stamping.Coils.In )
   END_RUNG wire#w3
   RUNG wire#powerrail
      Contact( "DEV_7".Convoyer.Modular_A.Pneumatics.Stamping.Coils.Out )
   END_RUNG wire#w3
   RUNG wire#powerrail
      I_Contact( "DEV_7".Convoyer.Modular_A.HMI.DoorDisable.BackDoor )
      I_Contact( "7A_DOOR_1" )
   END_RUNG wire#w4
   RUNG wire#powerrail
      I_Contact( "DEV_7".Convoyer.Modular_A.HMI.DoorDisable.FrontDoor )
      I_Contact( "7A_DOOR_2" )
   END_RUNG wire#w4
   RUNG wire#powerrail
      I_Contact( "DEV_7".Convoyer.Modular_A.HMI.DoorDisable.UnloadDoor )
      I_Contact( "7A_DOOR_3" )
   END_RUNG wire#w4
   RUNG wire#powerrail
      Contact( "7_BUTTON_RESET" )
   END_RUNG wire#w5
   RUNG wire#powerrail
      Contact( "7A_BUTTON_RESET_1" )
   END_RUNG wire#w5
   RUNG wire#powerrail
      Contact( "7A_BUTTON_RESET_2" )
   END_RUNG wire#w5
   // the same network as SCL:
   #Convoyer7A_Instance(InverterStatus := "Modular7A_SafetyStatus",   // "Convoyer7"
                        ESTOP := NOT "7A_ESTOP_1" OR NOT "7A_ESTOP_2" OR NOT "7_ESTOP" OR NOT "7_THERMOSTAT",
                        LIGHT_CURTAIN := NOT "7A_LIGHT_CURTAIN_1",
                        PROCES_STAMPING := "DEV_7".Convoyer.Modular_A.Pneumatics.Stamping.Coils.In OR "DEV_7".Convoyer.Modular_A.Pneumatics.Stamping.Coils.Out,
                        DOOR := (NOT "DEV_7".Convoyer.Modular_A.HMI.DoorDisable.BackDoor AND NOT "7A_DOOR_1") OR (NOT "DEV_7".Convoyer.Modular_A.HMI.DoorDisable.FrontDoor AND NOT "7A_DOOR_2") OR (NOT "DEV_7".Convoyer.Modular_A.HMI.DoorDisable.UnloadDoor AND NOT "7A_DOOR_3"),
                        FRQ_FEEDBACK := "7A_FRQ_SIG_1",
                        RESET := "7_BUTTON_RESET" OR "7A_BUTTON_RESET_1" OR "7A_BUTTON_RESET_2",
                        InverterControl => "Modula7A_SafetyControl",
                        SAFETY_OK => "DEV_7".Convoyer.Modular_A.Safety.SafetyOK,
                        INVERTER_OK => "DEV_7".Convoyer.Modular_A.Safety.InverterOK,
                        REQ_RESET_ESTOP => "DEV_7".Convoyer.Modular_A.Safety.REQ_RESET,
                        SAFETY_VALVE => "7A_Valve_Safety_1");
END_REGION

REGION Network 2
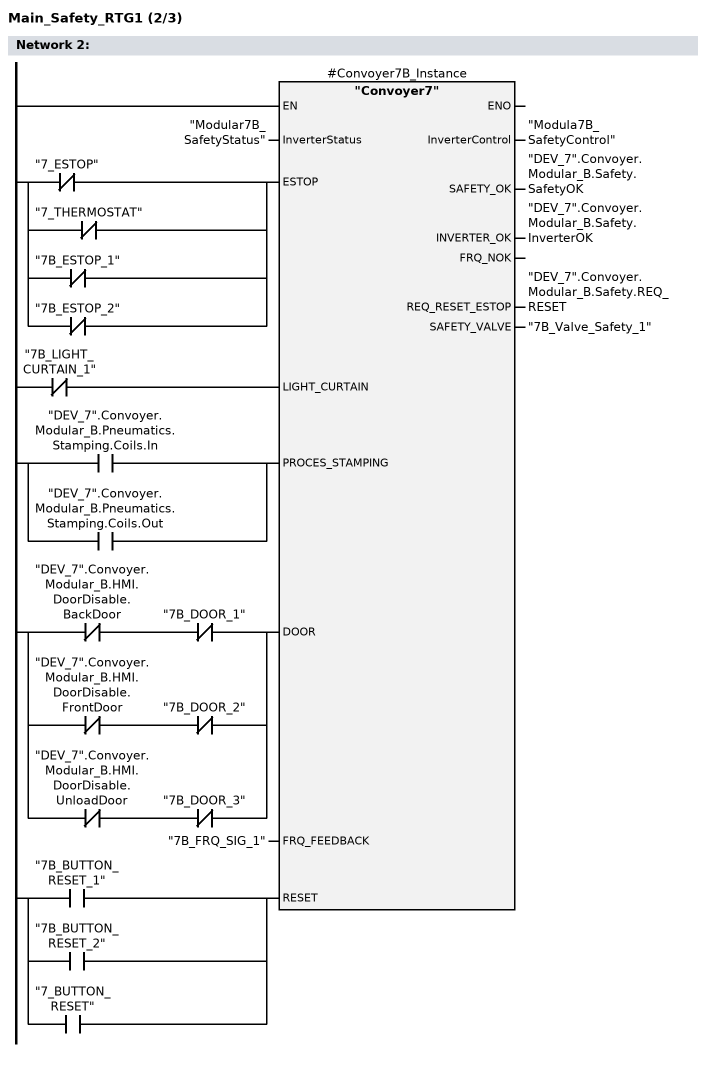
   RUNG wire#powerrail
      #Convoyer7B_Instance(ESTOP := wire#w1, LIGHT_CURTAIN := wire#w2, PROCES_STAMPING := wire#w3, DOOR := wire#w4, RESET := wire#w5, InverterStatus := "Modular7B_SafetyStatus", FRQ_FEEDBACK := "7B_FRQ_SIG_1", InverterControl => "Modula7B_SafetyControl", SAFETY_OK => "DEV_7".Convoyer.Modular_B.Safety.SafetyOK, INVERTER_OK => "DEV_7".Convoyer.Modular_B.Safety.InverterOK, FRQ_NOK =>, REQ_RESET_ESTOP => "DEV_7".Convoyer.Modular_B.Safety.REQ_RESET, SAFETY_VALVE => "7B_Valve_Safety_1")
   END_RUNG
   RUNG wire#powerrail
      I_Contact( "7_ESTOP" )
   END_RUNG wire#w1
   RUNG wire#powerrail
      I_Contact( "7_THERMOSTAT" )
   END_RUNG wire#w1
   RUNG wire#powerrail
      I_Contact( "7B_ESTOP_1" )
   END_RUNG wire#w1
   RUNG wire#powerrail
      I_Contact( "7B_ESTOP_2" )
   END_RUNG wire#w1
   RUNG wire#powerrail
      I_Contact( "7B_LIGHT_CURTAIN_1" )
   END_RUNG wire#w2
   RUNG wire#powerrail
      Contact( "DEV_7".Convoyer.Modular_B.Pneumatics.Stamping.Coils.In )
   END_RUNG wire#w3
   RUNG wire#powerrail
      Contact( "DEV_7".Convoyer.Modular_B.Pneumatics.Stamping.Coils.Out )
   END_RUNG wire#w3
   RUNG wire#powerrail
      I_Contact( "DEV_7".Convoyer.Modular_B.HMI.DoorDisable.BackDoor )
      I_Contact( "7B_DOOR_1" )
   END_RUNG wire#w4
   RUNG wire#powerrail
      I_Contact( "DEV_7".Convoyer.Modular_B.HMI.DoorDisable.FrontDoor )
      I_Contact( "7B_DOOR_2" )
   END_RUNG wire#w4
   RUNG wire#powerrail
      I_Contact( "DEV_7".Convoyer.Modular_B.HMI.DoorDisable.UnloadDoor )
      I_Contact( "7B_DOOR_3" )
   END_RUNG wire#w4
   RUNG wire#powerrail
      Contact( "7B_BUTTON_RESET_1" )
   END_RUNG wire#w5
   RUNG wire#powerrail
      Contact( "7B_BUTTON_RESET_2" )
   END_RUNG wire#w5
   RUNG wire#powerrail
      Contact( "7_BUTTON_RESET" )
   END_RUNG wire#w5
   // the same network as SCL:
   #Convoyer7B_Instance(InverterStatus := "Modular7B_SafetyStatus",   // "Convoyer7"
                        ESTOP := NOT "7_ESTOP" OR NOT "7_THERMOSTAT" OR NOT "7B_ESTOP_1" OR NOT "7B_ESTOP_2",
                        LIGHT_CURTAIN := NOT "7B_LIGHT_CURTAIN_1",
                        PROCES_STAMPING := "DEV_7".Convoyer.Modular_B.Pneumatics.Stamping.Coils.In OR "DEV_7".Convoyer.Modular_B.Pneumatics.Stamping.Coils.Out,
                        DOOR := (NOT "DEV_7".Convoyer.Modular_B.HMI.DoorDisable.BackDoor AND NOT "7B_DOOR_1") OR (NOT "DEV_7".Convoyer.Modular_B.HMI.DoorDisable.FrontDoor AND NOT "7B_DOOR_2") OR (NOT "DEV_7".Convoyer.Modular_B.HMI.DoorDisable.UnloadDoor AND NOT "7B_DOOR_3"),
                        FRQ_FEEDBACK := "7B_FRQ_SIG_1",
                        RESET := "7B_BUTTON_RESET_1" OR "7B_BUTTON_RESET_2" OR "7_BUTTON_RESET",
                        InverterControl => "Modula7B_SafetyControl",
                        SAFETY_OK => "DEV_7".Convoyer.Modular_B.Safety.SafetyOK,
                        INVERTER_OK => "DEV_7".Convoyer.Modular_B.Safety.InverterOK,
                        REQ_RESET_ESTOP => "DEV_7".Convoyer.Modular_B.Safety.REQ_RESET,
                        SAFETY_VALVE => "7B_Valve_Safety_1");
END_REGION

REGION Network 3
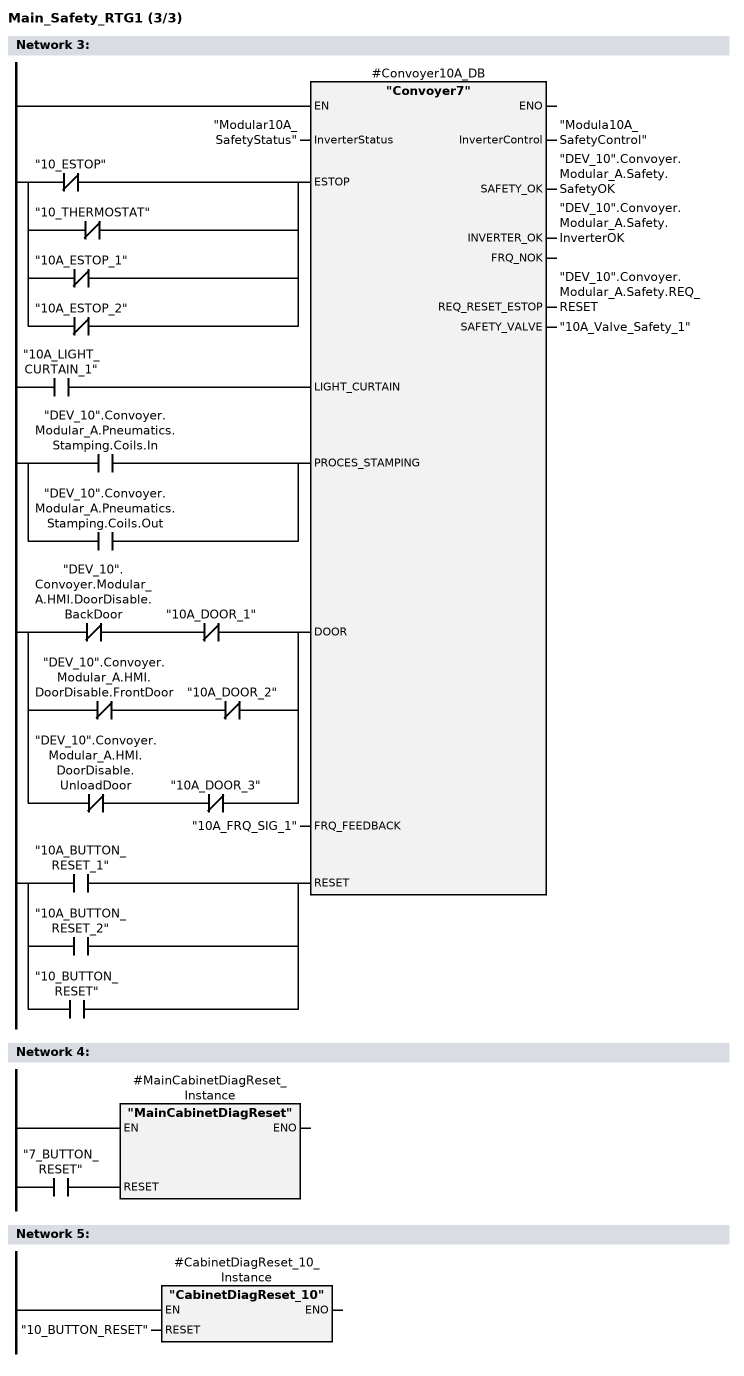
   RUNG wire#powerrail
      #Convoyer10A_DB(ESTOP := wire#w1, LIGHT_CURTAIN := wire#w2, PROCES_STAMPING := wire#w3, DOOR := wire#w4, RESET := wire#w5, InverterStatus := "Modular10A_SafetyStatus", FRQ_FEEDBACK := "10A_FRQ_SIG_1", InverterControl => "Modula10A_SafetyControl", SAFETY_OK => "DEV_10".Convoyer.Modular_A.Safety.SafetyOK, INVERTER_OK => "DEV_10".Convoyer.Modular_A.Safety.InverterOK, FRQ_NOK =>, REQ_RESET_ESTOP => "DEV_10".Convoyer.Modular_A.Safety.REQ_RESET, SAFETY_VALVE => "10A_Valve_Safety_1")
   END_RUNG
   RUNG wire#powerrail
      I_Contact( "10_ESTOP" )
   END_RUNG wire#w1
   RUNG wire#powerrail
      I_Contact( "10_THERMOSTAT" )
   END_RUNG wire#w1
   RUNG wire#powerrail
      I_Contact( "10A_ESTOP_1" )
   END_RUNG wire#w1
   RUNG wire#powerrail
      I_Contact( "10A_ESTOP_2" )
   END_RUNG wire#w1
   RUNG wire#powerrail
      Contact( "10A_LIGHT_CURTAIN_1" )
   END_RUNG wire#w2
   RUNG wire#powerrail
      Contact( "DEV_10".Convoyer.Modular_A.Pneumatics.Stamping.Coils.In )
   END_RUNG wire#w3
   RUNG wire#powerrail
      Contact( "DEV_10".Convoyer.Modular_A.Pneumatics.Stamping.Coils.Out )
   END_RUNG wire#w3
   RUNG wire#powerrail
      I_Contact( "DEV_10".Convoyer.Modular_A.HMI.DoorDisable.BackDoor )
      I_Contact( "10A_DOOR_1" )
   END_RUNG wire#w4
   RUNG wire#powerrail
      I_Contact( "DEV_10".Convoyer.Modular_A.HMI.DoorDisable.FrontDoor )
      I_Contact( "10A_DOOR_2" )
   END_RUNG wire#w4
   RUNG wire#powerrail
      I_Contact( "DEV_10".Convoyer.Modular_A.HMI.DoorDisable.UnloadDoor )
      I_Contact( "10A_DOOR_3" )
   END_RUNG wire#w4
   RUNG wire#powerrail
      Contact( "10A_BUTTON_RESET_1" )
   END_RUNG wire#w5
   RUNG wire#powerrail
      Contact( "10A_BUTTON_RESET_2" )
   END_RUNG wire#w5
   RUNG wire#powerrail
      Contact( "10_BUTTON_RESET" )
   END_RUNG wire#w5
   // the same network as SCL:
   #Convoyer10A_DB(InverterStatus := "Modular10A_SafetyStatus",   // "Convoyer7"
                   ESTOP := NOT "10_ESTOP" OR NOT "10_THERMOSTAT" OR NOT "10A_ESTOP_1" OR NOT "10A_ESTOP_2",
                   LIGHT_CURTAIN := "10A_LIGHT_CURTAIN_1",
                   PROCES_STAMPING := "DEV_10".Convoyer.Modular_A.Pneumatics.Stamping.Coils.In OR "DEV_10".Convoyer.Modular_A.Pneumatics.Stamping.Coils.Out,
                   DOOR := (NOT "DEV_10".Convoyer.Modular_A.HMI.DoorDisable.BackDoor AND NOT "10A_DOOR_1") OR (NOT "DEV_10".Convoyer.Modular_A.HMI.DoorDisable.FrontDoor AND NOT "10A_DOOR_2") OR (NOT "DEV_10".Convoyer.Modular_A.HMI.DoorDisable.UnloadDoor AND NOT "10A_DOOR_3"),
                   FRQ_FEEDBACK := "10A_FRQ_SIG_1",
                   RESET := "10A_BUTTON_RESET_1" OR "10A_BUTTON_RESET_2" OR "10_BUTTON_RESET",
                   InverterControl => "Modula10A_SafetyControl",
                   SAFETY_OK => "DEV_10".Convoyer.Modular_A.Safety.SafetyOK,
                   INVERTER_OK => "DEV_10".Convoyer.Modular_A.Safety.InverterOK,
                   REQ_RESET_ESTOP => "DEV_10".Convoyer.Modular_A.Safety.REQ_RESET,
                   SAFETY_VALVE => "10A_Valve_Safety_1");
END_REGION

REGION Network 4
   RUNG wire#powerrail
      #MainCabinetDiagReset_Instance(RESET := wire#w1)
   END_RUNG
   RUNG wire#powerrail
      Contact( "7_BUTTON_RESET" )
   END_RUNG wire#w1
   // the same network as SCL:
   #MainCabinetDiagReset_Instance(RESET := "7_BUTTON_RESET");   // "MainCabinetDiagReset"
END_REGION

REGION Network 5
   RUNG wire#powerrail
      #CabinetDiagReset_10_Instance(RESET := "10_BUTTON_RESET")
   END_RUNG
   // the same network as SCL:
   #CabinetDiagReset_10_Instance(RESET := "10_BUTTON_RESET");   // "CabinetDiagReset_10"
END_REGION
END_FUNCTION_BLOCK

FUNCTION_BLOCK "MitshubishiRobot"
{ S7_Optimized_Access := 'TRUE' }
VERSION : 0.1
   VAR_INPUT 
      Safety : Bool;
      Reset : Bool;
      RobotOutputData : "GeneralRobotOutputData";
   END_VAR

   VAR_OUTPUT 
      Status : "Status";
   END_VAR

   VAR_IN_OUT 
      Enable : Bool;
      RobotInputData : "GeneralRobotInputData";
   END_VAR

   VAR 
      state { S7_SetPoint := 'False'} : "s_changeState";
      R_TRIG_Safety {InstructionName := 'R_TRIG'; LibVersion := '1.0'} : R_TRIG;
      R_TRIG_RobotError {InstructionName := 'R_TRIG'; LibVersion := '1.0'} : R_TRIG;
   END_VAR

   VAR CONSTANT 
      S_IDLE : Int := 0;
      S_ERROR : Int := 10;
      S_BUSY : Int := 20;
   END_VAR


BEGIN
	//************************************************************
	//===Author: Mateusz Połojko
	//-----Linkedin: https://pl.linkedin.com/in/mateusz-po%C5%82ojko-52a3541b1
	//-----Github: https://github.com/Bhazel95
	//===Description:
	//-----Function block for sending + rvc commands/status of Mitsubishi robot
	//===Customer:
	//-----Apator Powogaz S.A.
	//************************************************************
	
	REGION R/F_TRIG
	    #R_TRIG_Safety(CLK:= NOT #Safety);
	    #R_TRIG_RobotError(CLK:=#RobotOutputData.Error);
	END_REGION
	
	CASE #state.state OF
	    #S_IDLE:
	        //Funkcja wejścia
	        IF #state.inputFlag AND NOT #state.outputFlag THEN
	            #state.name := 'IDLE';
	            #Status.Ready := TRUE;
	            #Status.Busy := FALSE;
	            #Status.Error := FALSE;
	        END_IF;
	        
	        //Funkcja cykliczna
	        IF NOT #state.inputFlag AND NOT #state.outputFlag THEN
	            IF #Enable THEN
	                #RobotInputData.Start := TRUE;
	            END_IF;
	            IF #RobotOutputData.DuringExecute AND #RobotOutputData.SequenceStarted THEN
	                #RobotInputData.Start := FALSE;
	                "changeState"(newState:=#S_BUSY,
	                              Data:=#state);
	            END_IF;
	        END_IF;
	        
	        //Funkcja wyjściowa 
	        IF #state.outputFlag THEN
	            ;
	        END_IF;
	        
	    #S_ERROR:
	        //Funkcja wejścia
	        IF #state.inputFlag AND NOT #state.outputFlag THEN
	            #state.name := 'ERROR';
	            #Status.Ready := FALSE;
	            #Status.Busy := FALSE;
	            #Status.Error := TRUE;
	        END_IF;
	        
	        //Funkcja cykliczna
	        IF NOT #state.inputFlag AND NOT #state.outputFlag THEN
	            IF #Safety AND #Reset AND NOT #RobotOutputData.Error THEN
	                #RobotInputData.Auto := TRUE;
	            END_IF;
	        END_IF;
	        
	        //Funkcja wyjściowa 
	        IF #state.outputFlag THEN
	            ;
	        END_IF;
	        
	    #S_BUSY:
	        //Funkcja wejścia
	        IF #state.inputFlag AND NOT #state.outputFlag THEN
	            #state.name := 'DURING_PROGRAM';
	            #Status.Ready := FALSE;
	            #Status.Busy := TRUE;
	            #Status.Error := FALSE;
	        END_IF;
	        
	        //Funkcja cykliczna
	        IF NOT #state.inputFlag AND NOT #state.outputFlag THEN
	            IF NOT #RobotOutputData.SequenceStarted THEN
	                "changeState"(newState := #S_IDLE,
	                              Data := #state);
	            END_IF;
	        END_IF;
	        
	        //Funkcja wyjściowa 
	        IF #state.outputFlag THEN
	            ;
	        END_IF;
	END_CASE;
	
	IF NOT #R_TRIG_Safety.Q OR #R_TRIG_RobotError.Q THEN
	    "changeState"(newState := #S_ERROR,
	                  Data := #state);
	END_IF;
	
	REGION Change state
	    IF #state.inputFlag AND NOT #state.outputFlag THEN
	        #state.inputFlag := FALSE;
	    END_IF;
	    #state.outputFlag := FALSE;
	END_REGION
END_FUNCTION_BLOCK

ORGANIZATION_BLOCK "Startup"
TITLE = "Complete Restart"
{ S7_Optimized_Access := 'TRUE' }
VERSION : 0.1

BEGIN
	REGION Motor
	    "DEV_7".Convoyer.Modular_A.MotorControl.MC_MOVEJOG.Velocity := 50;
	    "DEV_7".Convoyer.Modular_A.MotorControl.MC_MOVEJOG.Acceleration := 60;
	    "DEV_7".Convoyer.Modular_A.MotorControl.MC_MOVEJOG.Deceleration := 120;
	    
	    "DEV_7".Convoyer.Modular_B.MotorControl.MC_MOVEJOG.Velocity := 0.15;
	    "DEV_7".Convoyer.Modular_B.MotorControl.MC_MOVEJOG.Acceleration := 0.3;
	    "DEV_7".Convoyer.Modular_B.MotorControl.MC_MOVEJOG.Deceleration := 0.7;
	END_REGION
	REGION SKIP FIRST SOCKET
	    "ModularConvoyer_7A_DB".Local.isMoved := TRUE;
	    "ModularConvoyer_7B_DB".Local.isMoved := TRUE;
	    
	END_REGION
	
	
	
END_ORGANIZATION_BLOCK
